SUBAPPLICATION mapping_Buttons (* Subapplication Type *)
  (* Standard: 61499-2 *)
  (* Version 1.0, 2023-01-29, Franz *)
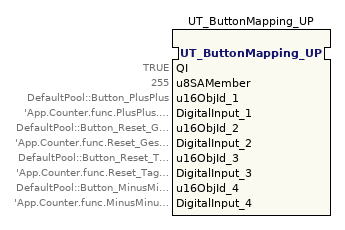
  FBS
    UT_ButtonMapping_UP : UT_ButtonMapping_UP(QI := TRUE, u8SAMember := 255, u16ObjId_1 := DefaultPool::Button_PlusPlus, DigitalInput_1 := 'App.Counter.func.PlusPlus.Button', u16ObjId_2 := DefaultPool::Button_Reset_Gesamtzaehler, DigitalInput_2 := 'App.Counter.func.Reset_Gesamtzaehler.Button', u16ObjId_3 := DefaultPool::Button_Reset_Tageszaehler, DigitalInput_3 := 'App.Counter.func.Reset_Tageszaehler.Button', u16ObjId_4 := DefaultPool::Button_MinusMinus, DigitalInput_4 := 'App.Counter.func.MinusMinus.Button');
  END_FBS
END_SUBAPPLICATION
